// TIA Portal V16 export
// export: Created 2024-12-03T15:41:44.1733403Z, ExportSetting WithDefaults, DisplayName Totally Integrated Automation Portal, DisplayVersion V16 Update 6, DisplayName TIA Portal Version Control Interface, DisplayVersion V16 Update 2, DisplayName TIA Portal Openness, DisplayVersion V16 Update 6, DisplayName TIA Portal Teamcenter Gateway, DisplayVersion V16, DisplayName SINAMICS Startdrive Advanced, DisplayVersion V16 Update 5, DisplayName SINAMICS Startdrive G130, G150, S120, S150, SINAMICS MV, S210, DisplayVersion V16 Update 5, DisplayName SINAMICS Startdrive G110M, G120, G120C, G120D, G120P, G115D, DisplayVersion V16 Update 5, DisplayName STEP 7 Professional, DisplayVersion V16 Update 6, DisplayName STEP 7 Safety, DisplayVersion V16, DisplayName WinCC Advanced / Unified PC, DisplayVersion V16 Update 6
DATA_BLOCK "Inputs_DB"   // DB1
{ S7_Optimized_Access := 'FALSE' }
VERSION : 0.1
// stored: AutoNumber true, DBAccessibleFromOPCUA true, IsOnlyStoredInLoadMemory false, IsWriteProtectedInAS false
   VAR
      AlwaysOff : "SmartBooldt";
      AlwaysOn : "SmartBooldt";
      Reset_System { S7_SetPoint := 'True'} : "SmartBooldt";
      EMG_OK { S7_SetPoint := 'True'} : "SmartBooldt";
      Fire_Alarm_Active { S7_SetPoint := 'True'} : "SmartBooldt";
      ToReplace { S7_SetPoint := 'True'} : "SmartBooldt";
      FTC_102_L2 { S7_SetPoint := 'True'} : "SmartBooldt";
      FTC_102_L4 { S7_SetPoint := 'True'} : "SmartBooldt";
      FTC_102_R2 { S7_SetPoint := 'True'} : "SmartBooldt";
      FTC_102_R4 { S7_SetPoint := 'True'} : "SmartBooldt";
      FTC_103_L2 { S7_SetPoint := 'True'} : "SmartBooldt";
      FTC_103_L4 { S7_SetPoint := 'True'} : "SmartBooldt";
      FTC_103_R2 { S7_SetPoint := 'True'} : "SmartBooldt";
      FTC_103_R4 { S7_SetPoint := 'True'} : "SmartBooldt";
      FTC_104_L2 { S7_SetPoint := 'True'} : "SmartBooldt";
      FTC_104_L4 { S7_SetPoint := 'True'} : "SmartBooldt";
      FTC_104_R2 { S7_SetPoint := 'True'} : "SmartBooldt";
      FTC_104_R4 { S7_SetPoint := 'True'} : "SmartBooldt";
      FTC_105_L2 { S7_SetPoint := 'True'} : "SmartBooldt";
      FTC_105_L4 { S7_SetPoint := 'True'} : "SmartBooldt";
      FTC_105_R2 { S7_SetPoint := 'True'} : "SmartBooldt";
      FTC_105_R4 { S7_SetPoint := 'True'} : "SmartBooldt";
      FTC_106_L2 { S7_SetPoint := 'True'} : "SmartBooldt";
      FTC_106_L4 { S7_SetPoint := 'True'} : "SmartBooldt";
      FTC_106_R2 { S7_SetPoint := 'True'} : "SmartBooldt";
      FTC_106_R4 { S7_SetPoint := 'True'} : "SmartBooldt";
      FTC_107_L2 { S7_SetPoint := 'True'} : "SmartBooldt";
      FTC_107_L4 { S7_SetPoint := 'True'} : "SmartBooldt";
      FTC_107_R2 { S7_SetPoint := 'True'} : "SmartBooldt";
      FTC_107_R4 { S7_SetPoint := 'True'} : "SmartBooldt";
      FTC_108_L2 { S7_SetPoint := 'True'} : "SmartBooldt";
      FTC_108_L4 { S7_SetPoint := 'True'} : "SmartBooldt";
      FTC_108_R2 { S7_SetPoint := 'True'} : "SmartBooldt";
      FTC_108_R4 { S7_SetPoint := 'True'} : "SmartBooldt";
      FTC_109_L2 { S7_SetPoint := 'True'} : "SmartBooldt";
      FTC_109_L4 { S7_SetPoint := 'True'} : "SmartBooldt";
      FTC_109_R2 { S7_SetPoint := 'True'} : "SmartBooldt";
      FTC_109_R4 { S7_SetPoint := 'True'} : "SmartBooldt";
      FTC_110_L2 { S7_SetPoint := 'True'} : "SmartBooldt";
      FTC_110_L4 { S7_SetPoint := 'True'} : "SmartBooldt";
      FTC_110_R2 { S7_SetPoint := 'True'} : "SmartBooldt";
      FTC_110_R4 { S7_SetPoint := 'True'} : "SmartBooldt";
      FTC_111_L2 { S7_SetPoint := 'True'} : "SmartBooldt";
      FTC_111_L4 { S7_SetPoint := 'True'} : "SmartBooldt";
      FTC_111_R2 { S7_SetPoint := 'True'} : "SmartBooldt";
      FTC_111_R4 { S7_SetPoint := 'True'} : "SmartBooldt";
      FTC_112_L2 { S7_SetPoint := 'True'} : "SmartBooldt";
      FTC_112_L4 { S7_SetPoint := 'True'} : "SmartBooldt";
      FTC_112_R2 { S7_SetPoint := 'True'} : "SmartBooldt";
      FTC_112_R4 { S7_SetPoint := 'True'} : "SmartBooldt";
      FTC_113_L2 { S7_SetPoint := 'True'} : "SmartBooldt";
      FTC_113_L4 { S7_SetPoint := 'True'} : "SmartBooldt";
      FTC_113_R2 { S7_SetPoint := 'True'} : "SmartBooldt";
      FTC_113_R4 { S7_SetPoint := 'True'} : "SmartBooldt";
      FTC_114_L2 { S7_SetPoint := 'True'} : "SmartBooldt";
      FTC_114_L4 { S7_SetPoint := 'True'} : "SmartBooldt";
      FTC_114_R2 { S7_SetPoint := 'True'} : "SmartBooldt";
      FTC_114_R4 { S7_SetPoint := 'True'} : "SmartBooldt";
      FTC_115_L2 { S7_SetPoint := 'True'} : "SmartBooldt";
      FTC_115_L4 { S7_SetPoint := 'True'} : "SmartBooldt";
      FTC_115_R2 { S7_SetPoint := 'True'} : "SmartBooldt";
      FTC_115_R4 { S7_SetPoint := 'True'} : "SmartBooldt";
      FTC_201_L4 { S7_SetPoint := 'True'} : "SmartBooldt";
      FTC_201_L2 { S7_SetPoint := 'True'} : "SmartBooldt";
      FTC_201_R2 { S7_SetPoint := 'True'} : "SmartBooldt";
      FTC_201_R4 { S7_SetPoint := 'True'} : "SmartBooldt";
      FTC_202_L2 { S7_SetPoint := 'True'} : "SmartBooldt";
      FTC_202_L4 { S7_SetPoint := 'True'} : "SmartBooldt";
      FTC_202_R2 { S7_SetPoint := 'True'} : "SmartBooldt";
      FTC_202_R4 { S7_SetPoint := 'True'} : "SmartBooldt";
      FTC_203_L2 { S7_SetPoint := 'True'} : "SmartBooldt";
      FTC_203_L4 { S7_SetPoint := 'True'} : "SmartBooldt";
      FTC_203_R2 { S7_SetPoint := 'True'} : "SmartBooldt";
      FTC_203_R4 { S7_SetPoint := 'True'} : "SmartBooldt";
      FTC_301_L2 { S7_SetPoint := 'True'} : "SmartBooldt";
      FTC_301_L4 { S7_SetPoint := 'True'} : "SmartBooldt";
      FTC_301_R2 { S7_SetPoint := 'True'} : "SmartBooldt";
      FTC_301_R4 { S7_SetPoint := 'True'} : "SmartBooldt";
      FTC_302_L2 { S7_SetPoint := 'True'} : "SmartBooldt";
      FTC_302_L4 { S7_SetPoint := 'True'} : "SmartBooldt";
      FTC_302_R2 { S7_SetPoint := 'True'} : "SmartBooldt";
      FTC_302_R4 { S7_SetPoint := 'True'} : "SmartBooldt";
      FTC_303_L2 { S7_SetPoint := 'True'} : "SmartBooldt";
      FTC_303_L4 { S7_SetPoint := 'True'} : "SmartBooldt";
      FTC_303_R2 { S7_SetPoint := 'True'} : "SmartBooldt";
      FTC_303_R4 { S7_SetPoint := 'True'} : "SmartBooldt";
      FTC_304_L2 { S7_SetPoint := 'True'} : "SmartBooldt";
      FTC_304_L4 { S7_SetPoint := 'True'} : "SmartBooldt";
      FTC_304_R2 { S7_SetPoint := 'True'} : "SmartBooldt";
      FTC_304_R4 { S7_SetPoint := 'True'} : "SmartBooldt";
      FTC_305_L2 { S7_SetPoint := 'True'} : "SmartBooldt";
      FTC_305_L4 { S7_SetPoint := 'True'} : "SmartBooldt";
      FTC_305_R2 { S7_SetPoint := 'True'} : "SmartBooldt";
      FTC_305_R4 { S7_SetPoint := 'True'} : "SmartBooldt";
      FTC_DRV_101_1_I1 { S7_SetPoint := 'True'} : "SmartBooldt";
      FTC_DRV_101_1_I2 { S7_SetPoint := 'True'} : "SmartBooldt";
      FTC_DRV_101_1_I3 { S7_SetPoint := 'True'} : "SmartBooldt";
      FTC_DRV_101_1_I4 { S7_SetPoint := 'True'} : "SmartBooldt";
      FTC_SKU_101_I1 { S7_SetPoint := 'True'} : "SmartBooldt";
      FTC_SKU_101_I2 { S7_SetPoint := 'True'} : "SmartBooldt";
   END_VAR
BEGIN
   AlwaysOn.State := true;
END_DATA_BLOCK
